Fanuc KAREL source: kb00077.KL

-- PROVISIONAL review KL for V940-1; original PC SHA256 b3789e5dc129f1cd39b888d86dbff0fb37205b110e7ebe208d627469436dc880
-- Incomplete behavior may be omitted. Consult companion uncertainty JSON. Do not deploy.
PROGRAM KB00077
%NOLOCKGROUP
BEGIN
  -- V9_ZERO_TABLE_METADATA_HINT layout=0002_ascii; no indexed target words; source/name/runtime held
  -- UNRESOLVED_PC offsets 5-14; opcodes 3F,75
  -- UNRESOLVED_PC offsets 19-26; opcodes 9D,23
  -- UNRESOLVED_PC offsets 31-38; opcodes 9D,23
  -- UNRESOLVED_PC offsets 43-52; opcodes 3F,75
  -- UNRESOLVED_PC offsets 57-64; opcodes 9D,23
  -- UNRESOLVED_PC offsets 69-107; opcodes 27,22,2A,22,22,22,2A,22,31
  -- UNRESOLVED_PC offsets 112-116; opcodes 7F
END KB00077
